// TIA Portal V17 export
// export: Created 2025-03-05T08:03:05.5190104Z, ExportSetting WithDefaults, DisplayName Totally Integrated Automation Portal, DisplayVersion V17 Update 8, DisplayName TIA Portal Openness, DisplayVersion V17 Update 8, DisplayName TIA Portal Version Control Interface, DisplayVersion V17, DisplayName SINAMICS Startdrive Advanced, DisplayVersion V17 SP2, DisplayName SINAMICS Startdrive G110M, G120, G120C, G120D, G120P, G115D, DisplayVersion V17 SP2, DisplayName SINAMICS Startdrive G130, G150, S120, S150, SINAMICS MV, S210, DisplayVersion V17 SP2, DisplayName STEP 7 Professional, DisplayVersion V17 Update 8, DisplayName SINUMERIK ONE STEP 7 Toolbox, DisplayVersion V17 Update 12, DisplayName SINUMERIK 840D sl STEP 7 Toolbox, DisplayVersion V17 Update 12, DisplayName STEP 7 Safety, DisplayVersion V17 Update 6, DisplayName WinCC Advanced, DisplayVersion V17 Update 8
DATA_BLOCK "DB21013_PF_1_HOPPERS_UNIT_01"   // DB21013
VERSION : 0.1
// stored: AutoNumber false, DBAccessibleFromOPCUA true, DBAccessibleFromWebserver true, InstanceOfName FB21013_POWDER_FEEDER_HOPPER, InstanceOfType FB
"FB21013_POWDER_FEEDER_HOPPER"
   // VAR_INPUT
   //    OPTIONS_0 : Byte;
   //    iGENERAL_CONDITIONS : Bool;
   //    iPF_LINE_1_NOT_READY_FAULT : Bool;
   //    iPF_PROFINET_MODE_ACTIVE_FAULT_LINE_1 : Bool;
   //    iPF_LINE_2_NOT_READY_FAULT : Bool;
   //    iMANUAL_START_REQ_LINE_1 : Bool;
   //    iMANUAL_START_REQ_LINE_2 : Bool;
   //    iMANUAL_STOP_REQ_LINE_1 : Bool;
   //    iMANUAL_STOP_REQ_LINE_2 : Bool;
   //    iPF_INTERLOCK_INPUTS : "POWDER FEEDER INTERLOCK INPUT";
   //    iFEEDER_PROFINET_MODE_ACTIVE : Bool;
   //    iCONTROL_ON_DELAYED : Bool;
   //    iAUTO_START_REQUEST : Bool;
   //    iAUTO_STOP_REQUEST : Bool;
   //    iHMI_GAS_SETPOINT_L1 : Real;
   //    iHMI_GAS_SETPOINT_L2 : Real;
   //    iHMI_DISK_SETPOINT_L1 : Real;
   //    iHMI_DISK_SETPOINT_L2 : Real;
   //    iCNC_GAS_SETPOINT_L1 : Real;
   //    iCNC_GAS_SETPOINT_L2 : Real;
   //    iCNC_DISK_SETPOINT_L1 : Real;
   //    iCNC_DISK_SETPOINT_L2 : Real;
   //    iFEEDER_PLC_AUX_VALUES : "POWDER FEEDER PLC AUXILIAR";
   // END_VAR
   // VAR_OUTPUT
   //    oSTATION_IS_ALARMS : Bool;
   //    oSTATION_WARNINGS : Bool;
   //    o_fShutdownToPF_Line1 { ExternalAccessible := 'False'; ExternalVisible := 'False'; ExternalWritable := 'False'} : Bool;
   //    o_fShutdownToPF_Line2 { ExternalAccessible := 'False'; ExternalVisible := 'False'; ExternalWritable := 'False'} : Bool;
   //    o_fFeedingAllOnCmd_Line1 { ExternalAccessible := 'False'; ExternalVisible := 'False'; ExternalWritable := 'False'} : Bool;
   //    o_fFeedingAllOnCmd_Line2 { ExternalAccessible := 'False'; ExternalVisible := 'False'; ExternalWritable := 'False'} : Bool;
   //    o_fCarriergasOnCmd_Line1 { ExternalAccessible := 'False'; ExternalVisible := 'False'; ExternalWritable := 'False'} : Bool;
   //    o_fCarriergasOnCmd_Line2 { ExternalAccessible := 'False'; ExternalVisible := 'False'; ExternalWritable := 'False'} : Bool;
   //    o_fFeedingAllOffCmd_Line1 { ExternalAccessible := 'False'; ExternalVisible := 'False'; ExternalWritable := 'False'} : Bool;
   //    o_fFeedingAllOffCmd_Line2 { ExternalAccessible := 'False'; ExternalVisible := 'False'; ExternalWritable := 'False'} : Bool;
   //    o_fCarriergasOffCmd_Line1 { ExternalAccessible := 'False'; ExternalVisible := 'False'; ExternalWritable := 'False'} : Bool;
   //    o_fCarriergasOffCmd_Line2 { ExternalAccessible := 'False'; ExternalVisible := 'False'; ExternalWritable := 'False'} : Bool;
   //    oALARM_POWDER_LINE_1_CLOGGED : Bool;
   //    oALARM_GAS_FLOW_BELOW_LOW_LIMIT_LN_1 : Bool;
   //    oALARM_DISK_SPEED_BELOW_LOW_LIMIT_LN_1 : Bool;
   //    oALARM_STIRRER_SPEED_BELOW_LOW_LIMIT_LN_1 : Bool;
   //    oALARM_GAS_FLOW_ABOVE_HIGH_LIMIT_LN_1 : Bool;
   //    oALARM_DISK_SPEED_ABOVE_HIGH_LIMIT_LN_1 : Bool;
   //    oALARM_STIRRER_SPEED_ABOVE_HIGH_LIMIT_LN_1 : Bool;
   //    oALARM_CARRIER_GAS_INLET_PRESSURE_TOO_LOW_LN_1 : Bool;
   //    oALARM_DISK_MOTOR_PLUGGED_IN_AND_READY_LN_1 : Bool;
   //    oALARM_STIRRER_PLUGGED_IN_AND_READY_LN_1 : Bool;
   //    oALARM_COMMUNICATION_RUNNING_LN_1 : Bool;
   //    oALARM_FEEDER_NOT_READY_LN_1 : Bool;
   //    oWARNING_GAS_FLOW_UNDER_LIMIT_LN_1 : Bool;
   //    oWARNING_DISK_SPEED_UNDER_LIMIT_LN_1 : Bool;
   //    oWARNING_STIRRER_SPEED_UNDER_LIMIT_LN_1 : Bool;
   //    oWARNING_GAS_FLOW_OVER_LIMIT_LN_1 : Bool;
   //    oWARNING_DISK_SPEED_OVER_LIMIT_LN_1 : Bool;
   //    oWARNING_STIRRER_SPEED_OVER_LIMIT_LN_1 : Bool;
   //    oALARM_POWDER_LINE_2_CLOGGED : Bool;
   //    oALARM_GAS_FLOW_BELOW_LOW_LIMIT_LN_2 : Bool;
   //    oALARM_DISK_SPEED_BELOW_LOW_LIMIT_LN_2 : Bool;
   //    oALARM_STIRRER_SPEED_BELOW_LOW_LIMIT_LN_2 : Bool;
   //    oALARM_GAS_FLOW_ABOVE_HIGH_LIMIT_LN_2 : Bool;
   //    oALARM_DISK_SPEED_ABOVE_HIGH_LIMIT_LN_2 : Bool;
   //    oALARM_STIRRER_SPEED_ABOVE_HIGH_LIMIT_LN_2 : Bool;
   //    oALARM_CARRIER_GAS_INLET_PRESSURE_TOO_LOW_LN_2 : Bool;
   //    oALARM_DISK_MOTOR_PLUGGED_IN_AND_READY_LN_2 : Bool;
   //    oALARM_STIRRER_PLUGGED_IN_AND_READY_LN_2 : Bool;
   //    oALARM_COMMUNICATION_RUNNING_LN_2 : Bool;
   //    oALARM_FEEDER_NOT_READY_LN_2 : Bool;
   //    oWARNING_GAS_FLOW_UNDER_LIMIT_LN_2 : Bool;
   //    oWARNING_DISK_SPEED_UNDER_LIMIT_LN_2 : Bool;
   //    oWARNING_STIRRER_SPEED_UNDER_LIMIT_LN_2 : Bool;
   //    oWARNING_GAS_FLOW_OVER_LIMIT_LN_2 : Bool;
   //    oWARNING_DISK_SPEED_OVER_LIMIT_LN_2 : Bool;
   //    oWARNING_STIRRER_SPEED_OVER_LIMIT_LN_2 : Bool;
   // END_VAR
   // VAR RETAIN
   //    DATA : "POWDER FEEDER HOPPER";
   //    INPUT_SETTINGS : Struct
   //       UNIT_NUMBER : Int;
   //       FEEDER_NUMBER : Int;
   //    END_STRUCT;
   //    Fault_timer { S7_SetPoint := 'True'} : TON_TIME;
   //    START_DONE_LINE_1 { S7_SetPoint := 'True'} : Bool;
   //    START_DONE_LINE_2 { S7_SetPoint := 'True'} : Bool;
   //    STOP_SEQUENCE_ON { S7_SetPoint := 'True'} : Bool;
   //    STOP_PULSE_LINE_1 : Bool;
   //    STOP_PULSE_LINE_2 : Bool;
   //    HOPPER_STATUS_LINE_1 : Byte;
   //    HOPPER_STATUS_LINE_2 : Byte;
   //    SWITCH_ON_SEQUENCE_LINE_1 : "FB21250_POWDER_ON_OFF_SEQUENCE";
   //    SWITCH_ON_SEQUENCE_LINE_2 : "FB21250_POWDER_ON_OFF_SEQUENCE";
   //    SWITCH_OFF_SEQUENCE_LINE_1 : "FB21250_POWDER_ON_OFF_SEQUENCE";
   //    SWITCH_OFF_SEQUENCE_LINE_2 : "FB21250_POWDER_ON_OFF_SEQUENCE";
   //    SWITCH_OFF_DELAY_LINE_1 { S7_SetPoint := 'True'} : TOF_TIME;
   //    SWITCH_OFF_DELAY_LINE_2 { S7_SetPoint := 'True'} : TOF_TIME;
   // END_VAR
BEGIN
END_DATA_BLOCK
